{attribute 'qualified_only'}
{attribute 'strict'}
{attrivute 'to_string'}
// Rolling interval to create a new log file when expired. 
TYPE E_RollingInterval :
(
	None,
	Hourly,
	Daily,
	Monthly
);
END_TYPE

(* stored: Version 1.1.0.1, ProductVersion 3.1.4024.4
   DUT E_RollingInterval: Id {6307f971-7bf8-46ec-9b38-ec512e24283a} *)
